TYPE WaferRecipe :
STRUCT
	Name : T_MaxString;
	InspectionType : InspectionTypes;
	MaxWaferHeightFromBase : UDINT;
	MinWaferHeightFromBase : UDINT;
	PassingWaferCavityPercentage : UDINT;
	MaxNumberFailedBarsAllowed : UINT;
END_STRUCT
END_TYPE

(* stored: Version 1.1.0.1
   DUT WaferRecipe: Id {1bb3a427-2311-4152-b1ad-99d63dfaf4f2} *)
